(*********************************** G.D S.p.A. - Technical Department ***********************************
============= PROGRAM INFO ============
FOLDER:             TBD
MACHINES INVOLVED:  TBD 

============= DESCRIPTION =============
csp - Downstream Interface

============= REVISIONS ===============
Date		Version	 	Author      	Description             
----------	-------		------------  	--------------------------------------------
2019/10/07 	0000.00	 	W. Gerstner		Creation of the PRG

**********************************************************************************************************)
(*$R
	process_ref := prc;
$*)
PROGRAM csp_main_interface_downstream
VAR
	prc:					process;
	prc_path:				STRING;	

END_VAR

_read_var_input();

_object_manager();

IF NOT objects_running()
THEN
	RETURN;	
END_IF

_read_process_image();

_mode_manager();

CASE process_get_mode(prc) of
	MODE_ABSENT,
	MODE_INACTIVE:
		RETURN;
	MODE_TEST:
		_handle_process_test();
END_CASE

_set_runtime_properties();

(********************************* BODY *********************************)

(************************************************************************)

_handle_messages();

_write_output();

ACTION _handle_messages:
;
END_ACTION

ACTION _handle_process_test:
;
END_ACTION

ACTION _mode_manager:
IF process_mode_req_is_pending(prc)
THEN
    process_apply_mode_req_first_step(prc);
    CASE process_get_mode(prc) OF
        MODE_TO_ABSENT:
			;
        MODE_TO_INACTIVE:
			;
        MODE_TO_TEST:
			;
        MODE_TO_OPERATIONAL:
			;
    END_CASE
    process_apply_mode_req_second_step(prc);
END_IF
END_ACTION

ACTION _object_manager:
IF objects_initialization()
THEN
	sub_process_init(
		object_name						:= 'csp_main_interface_downstream.prc', 
		process							:= csp_main_interface.prc, 
		CONVERSION_this					:= prc);
		
	prc_path 							:= process_get_path(prc);
END_IF

IF objects_running()
THEN
	process_cycle(prc);
END_IF
END_ACTION

ACTION _read_process_image:
;
END_ACTION

ACTION _read_var_input:
;
END_ACTION

ACTION _set_runtime_properties:
;
END_ACTION

ACTION _write_output:
;
END_ACTION

END_PROGRAM

(* stored: Version 1.1.0.1, ProductVersion 3.1.4022.12
   POU csp_main_interface_downstream: Id {e690a02a-a3a0-4399-ac03-6d4304fe5c06}, SpecialFunc None
   Action _handle_messages: Id {2b3814c4-e11c-46c9-887e-936e1aa03ff5}
   Action _handle_process_test: Id {d4adb3bf-a574-4607-8fdb-7de6430c4baa}
   Action _mode_manager: Id {16bd3b27-9969-4014-9bd0-2d095af906b3}
   Action _object_manager: Id {7d6f6353-6765-4d0c-8036-5ae58a077950}
   Action _read_process_image: Id {bf709767-1d60-41d5-bd1e-ffa40145115a}
   Action _read_var_input: Id {3c780d31-a324-4bdc-8edd-b657ae54e40c}
   Action _set_runtime_properties: Id {138749b3-27fc-48c1-8c49-4966d17d31a4}
   Action _write_output: Id {2f242421-eeb2-40f3-bd32-0b5886c8040a} *)
